// SIMATIC S7-200 project (STEP 7-Micro/WIN), CPU 224 CN REL 02.01

ORGANIZATION_BLOCK 主程序:OB1
TITLE=程序注释
BEGIN
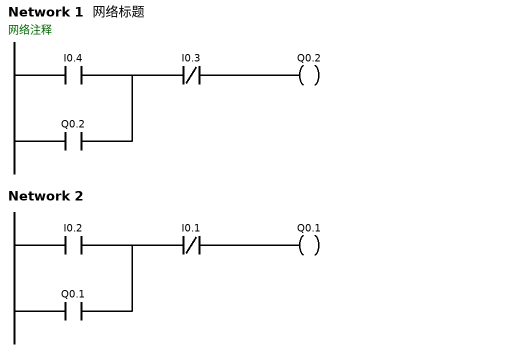
Network 1 // 网络标题
// 网络注释
LD     I0.4
O      Q0.2
AN     I0.3
=      Q0.2
Network 2
LD     I0.2
O      Q0.1
AN     I0.1
=      Q0.1
END_ORGANIZATION_BLOCK
